# EPICS autosave request: ADQImaging/iocs/qimageIOC/iocBoot/iocQImage/auto_settings.req
file "qimaging_settings.req",     P=$(P),  R=cam1:
file "NDStdArrays_settings.req",  P=$(P),  R=image1:
file "commonPlugin_settings.req", P=$(P)
